Staubli VAL3: test.pjx

--- test.pjx ---
Parameters version=s7.6.2 stackSize=5000 millimeterUnit=true
Program file=start.pgx
Program file=stop.pgx
Data file=test.dtx

--- test.dtx ---
mdesc mNomSpeed
pointRx safe = {x=-473.709167, y=42.287889, z=-99.734082, rx=-0.003569, ry=179.995424, rz=-0.000555, fatherId=world[0]}
pointRx work = {x=-473.709315, y=42.287111, z=-157.528576, rx=-0.003461, ry=179.99482, rz=-0.000845, fatherId=world[0]}
